# EPICS autosave request: ADPixirad/pixiradApp/Db/pixirad_settings.req
$(P)$(R)Threshold1
$(P)$(R)Threshold2
$(P)$(R)Threshold3
$(P)$(R)Threshold4
$(P)$(R)HVValue
$(P)$(R)HVState
$(P)$(R)HVMode
$(P)$(R)SyncInPolarity
$(P)$(R)SyncOutPolarity
$(P)$(R)SyncOutFunction
$(P)$(R)CoolingState
